FUNCTION F_4Args : INT
VAR_INPUT
    a : INT;
    b : INT;
    c : INT;
    d : INT;
END_VAR

F_4Args := a + b + c + d;

END_FUNCTION

(* stored: Version 1.1.0.1, ProductVersion 3.1.4024.16
   POU F_4Args: Id {6bde4f3e-6453-454d-b420-343d56666e26}, SpecialFunc None *)
